SYSTEM FLASHERW_TESTR (* Test FLASHERW on Remote Device *)
  (* Standard: 61499-1; Classification: Test; Type: SNAP Test *)
  (* Version 0.1, 2007-11-09, JHC, Holobloc Inc, Modified UDP addresses to work with WXP. *)
  (* Version 0.0, 2003-07-12, JHC, Rockwell Automation, Modified from RMT_DEV_TEST. *)
  APPLICATION TEST1 (* FB_ADD_INT test *)
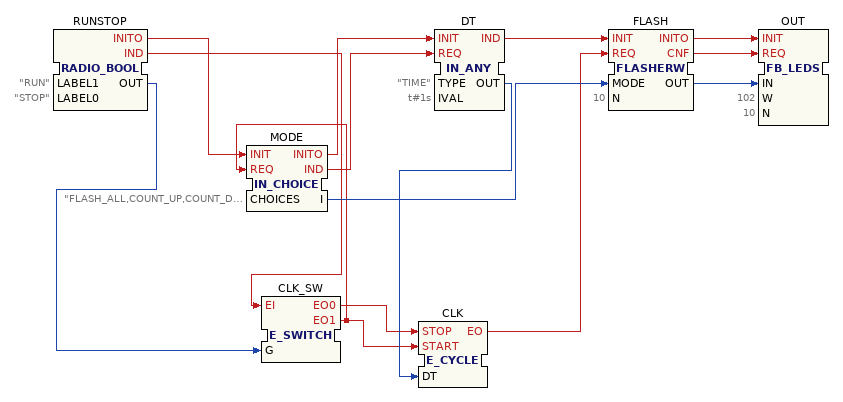
    FBS
      RUNSTOP : RADIO_BOOL(LABEL1 := "RUN", LABEL0 := "STOP");
      MODE : IN_CHOICE(CHOICES := "FLASH_ALL,COUNT_UP,COUNT_DOWN,CHASE_UP,CHASE_DOWN");
      DT : IN_ANY(TYPE := "TIME", IVAL := t#1s);
      CLK_SW : E_SWITCH;
      CLK : E_CYCLE;
      FLASH : FLASHERW(N := 10);
      OUT : FB_LEDS(W := 102, N := 10);
    END_FBS
    EVENT_CONNECTIONS
      RUNSTOP.INITO TO MODE.INIT;
      MODE.INITO TO DT.INIT;
      RUNSTOP.IND TO CLK_SW.EI;
      CLK_SW.EO0 TO CLK.STOP;
      CLK_SW.EO1 TO MODE.REQ;
      CLK_SW.EO1 TO CLK.START;
      MODE.IND TO DT.REQ;
      DT.IND TO FLASH.INIT;
      CLK.EO TO FLASH.REQ;
      FLASH.INITO TO OUT.INIT;
      FLASH.CNF TO OUT.REQ;
    END_CONNECTIONS
    DATA_CONNECTIONS
      MODE.I TO FLASH.MODE;
      DT.OUT TO CLK.DT;
      RUNSTOP.OUT TO CLK_SW.G;
      FLASH.OUT TO OUT.IN;
    END_CONNECTIONS
  END_APPLICATION
  DEVICE DEV_TESTER : FRAME_DEVICE(BOUNDS := [50,50,190,150], GRID := [1,1])
    RESOURCE RES2 : PANEL_RESOURCE
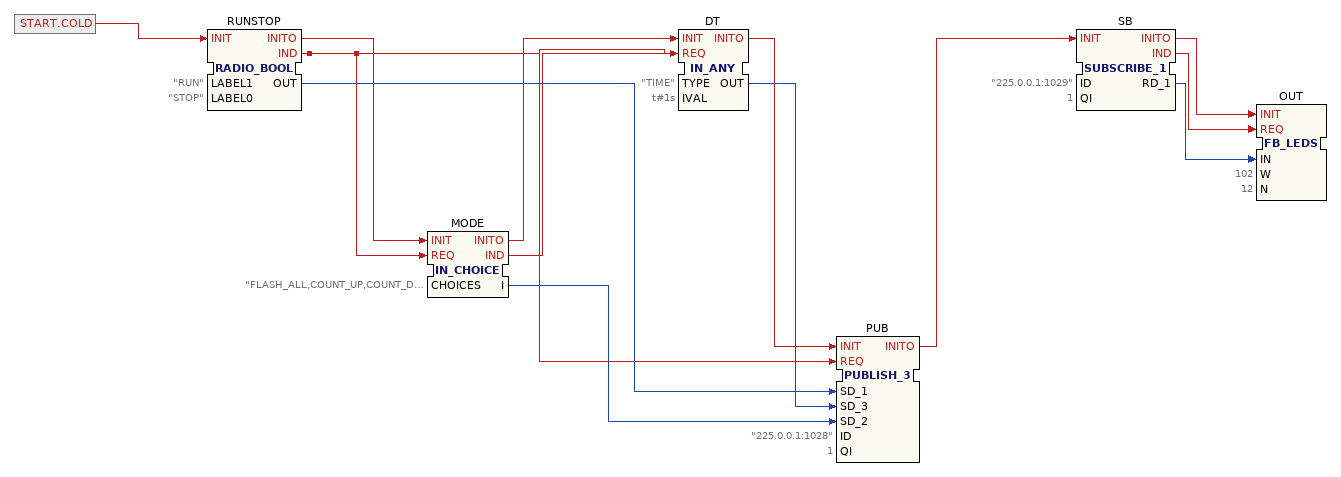
      FBS
        PUB : PUBLISH_3(ID := "225.0.0.1:1028", QI := 1);
        SB : SUBSCRIBE_1(ID := "225.0.0.1:1029", QI := 1);
        RUNSTOP : RADIO_BOOL(LABEL1 := "RUN", LABEL0 := "STOP");
        MODE : IN_CHOICE(CHOICES := "FLASH_ALL,COUNT_UP,COUNT_DOWN,CHASE_UP,CHASE_DOWN");
        DT : IN_ANY(TYPE := "TIME", IVAL := t#1s);
        OUT : FB_LEDS(W := 102, N := 12);
      END_FBS
      EVENT_CONNECTIONS
        PUB.INITO TO SB.INIT;
        RUNSTOP.INITO TO MODE.INIT;
        MODE.INITO TO DT.INIT;
        MODE.IND TO DT.REQ;
        START.COLD TO RUNSTOP.INIT;
        DT.INITO TO PUB.INIT;
        SB.INITO TO OUT.INIT;
        RUNSTOP.IND TO MODE.REQ;
        RUNSTOP.IND TO DT.REQ;
        RUNSTOP.IND TO PUB.REQ;
        SB.IND TO OUT.REQ;
      END_CONNECTIONS
      DATA_CONNECTIONS
        RUNSTOP.OUT TO PUB.SD_1;
        DT.OUT TO PUB.SD_3;
        SB.RD_1 TO OUT.IN;
        MODE.I TO PUB.SD_2;
      END_CONNECTIONS
    END_RESOURCE
  END_DEVICE
  DEVICE DEV1 : RMT_DEV(MGR_ID := "192.168.1.5:61499")
    RESOURCE RES2 : EMB_RES
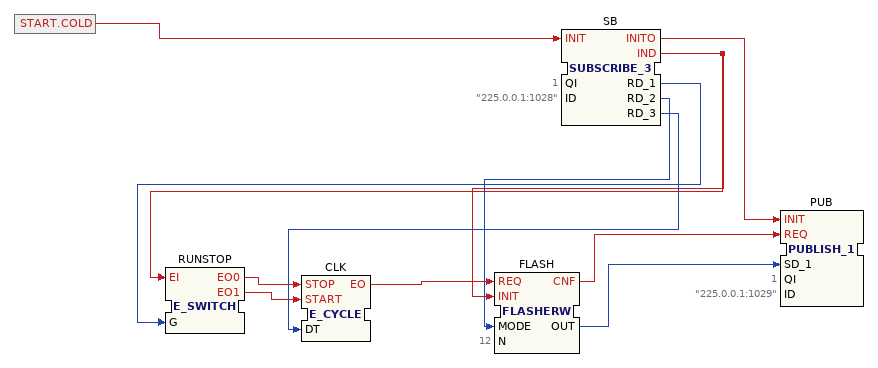
      FBS
        SB : SUBSCRIBE_3(QI := 1, ID := "225.0.0.1:1028");
        RUNSTOP : E_SWITCH;
        CLK : E_CYCLE;
        PUB : PUBLISH_1(QI := 1, ID := "225.0.0.1:1029");
        FLASH : FLASHERW(N := 12);
      END_FBS
      EVENT_CONNECTIONS
        SB.INITO TO PUB.INIT;
        SB.IND TO RUNSTOP.EI;
        RUNSTOP.EO0 TO CLK.STOP;
        RUNSTOP.EO1 TO CLK.START;
        CLK.EO TO FLASH.REQ;
        SB.IND TO FLASH.INIT;
        FLASH.CNF TO PUB.REQ;
        START.COLD TO SB.INIT;
      END_CONNECTIONS
      DATA_CONNECTIONS
        SB.RD_1 TO RUNSTOP.G;
        SB.RD_2 TO FLASH.MODE;
        SB.RD_3 TO CLK.DT;
        FLASH.OUT TO PUB.SD_1;
      END_CONNECTIONS
    END_RESOURCE
    RESOURCE MGR : RMT_RES
    END_RESOURCE
  END_DEVICE
  MAPPINGS
    TEST1.IN1 ON DEV_TESTER.RES1.IN1;
    TEST1.PLUS ON DEV_TESTER.RES1.PLUS;
    TEST1.IN2 ON DEV_TESTER.RES1.IN2;
    TEST1.EQUALS ON DEV_TESTER.RES1.EQUALS;
    TEST1.AD ON DEV1.RES1.AD;
    TEST2.RUNSTOP ON DEV_TESTER.RES2.RUNSTOP;
    TEST2.RESET ON DEV_TESTER.RES2.RESET;
    TEST2.PV ON DEV_TESTER.RES2.PV;
    TEST2.DT ON DEV_TESTER.RES2.DT;
    TEST2.RSSW ON DEV1.RES2.RUNSTOP;
    TEST2.CLK ON DEV1.RES2.CLK;
    TEST2.CTR ON DEV1.RES2.CTR;
    TEST2.Q ON DEV_TESTER.RES2.Q;
    TEST2.CV ON DEV_TESTER.RES2.CV;
    TEST1.RUNSTOP ON DEV_TESTER.RES2.RUNSTOP;
    TEST1.MODE ON DEV_TESTER.RES2.MODE;
    TEST1.DT ON DEV_TESTER.RES2.DT;
    TEST1.OUT ON DEV_TESTER.RES2.OUT;
  END_MAPPINGS
END_SYSTEM
